(* IEC 61131-3 sources: RegAx/test, 7 files *)

(* ---- Assert.st ---- *)
USING AxUnit.ResultFunctions;
USING System.Strings;

NAMESPACE AxUnit.Assert

    /// Succeeds when the provided condition is TRUE.
    FUNCTION PUBLIC IsTrue
        VAR_INPUT
            /// Condition that must evaluate to TRUE.
            condition : BOOL;
        END_VAR
        IF condition THEN
            axunit_Succeed();
        ELSE
            axunit_Fail('Condition is not true');
        END_IF;
    END_FUNCTION

    /// Succeeds when the provided condition is FALSE.
    FUNCTION PUBLIC IsFalse
        VAR_INPUT
            /// Condition that must evaluate to FALSE.
            condition : BOOL;
        END_VAR
        IF NOT condition THEN
            axunit_Succeed();
        ELSE
            axunit_Fail('Condition is not false');
        END_IF;
    END_FUNCTION

END_NAMESPACE

(* ---- TestRegexClasses.st ---- *)
USING AxUnit.Assert;
USING Simatic.Ax.RegAx;
NAMESPACE RegexTests

    {TestFixture}
    /// Verifies shorthand character classes like \d and \w.
    CLASS TestRegexClasses
        VAR
            /// Regex instance reused across class test cases.
            _regex : Regex;
        END_VAR

        {Test}
        /// Ensures one or more digits are matched by \d+.
        METHOD PUBLIC Matches_Digit_Class_With_Plus
            _regex.SetPattern('^\d+$$');
            _regex.SetInput('12345');

            IsTrue(_regex.Match());
            Equal(expected := '12345', actual := _regex.GetMatch());
        END_METHOD

        {Test}
        /// Ensures \d+ rejects inputs containing letters.
        METHOD PUBLIC Rejects_Digit_Class_When_Letters_Appear
            _regex.SetPattern('^\d+$$');
            _regex.SetInput('123a');

            IsFalse(_regex.Match());
        END_METHOD

        {Test}
        /// Ensures \w works together with a bounded range quantifier.
        METHOD PUBLIC Matches_Word_Class_With_Range_Quantifier
            _regex.SetPattern('^\w{3,5}$$');
            _regex.SetInput('ab_9');

            IsTrue(_regex.Match());
            Equal(expected := 'ab_9', actual := _regex.GetMatch());
        END_METHOD

        {Test}
        /// Ensures \w range quantifiers reject inputs below the minimum length.
        METHOD PUBLIC Rejects_Word_Class_When_Too_Short
            _regex.SetPattern('^\w{3,5}$$');
            _regex.SetInput('ab');

            IsFalse(_regex.Match());
        END_METHOD

        {Test}
        /// Ensures mixed alphabetic ranges like [a-zA-Z] match upper and lower case letters.
        METHOD PUBLIC Matches_Alphabetic_Character_Class_Range
            _regex.SetPattern('^[a-zA-Z]+$$');
            _regex.SetInput('AbCdEf');

            IsTrue(_regex.Match());
            Equal(expected := 'AbCdEf', actual := _regex.GetMatch());
        END_METHOD
    END_CLASS

END_NAMESPACE

(* ---- TestRegexEscapes.st ---- *)
USING AxUnit.Assert;
USING Simatic.Ax.RegAx;
USING System.Strings;
NAMESPACE RegexTests

    {TestFixture}
    /// Verifies escaped literals and IP-like matching scenarios.
    CLASS TestRegexEscapes
        VAR
            /// Regex instance reused across escape and IP test cases.
            _regex : Regex;
        END_VAR

        /// Returns the substring after the first occurrence of a separator.
        METHOD PRIVATE TailAfterFirstSeparator : STRING
            VAR_INPUT
                input : STRING;
                separator : CHAR;
            END_VAR
            VAR
                currentIndex : INT;
                inputLength : INT;
                result : STRING;
                separatorFound : BOOL;
            END_VAR

            result := '';
            inputLength := LengthOf(input);
            separatorFound := FALSE;

            FOR currentIndex := 1 TO inputLength DO
                IF separatorFound THEN
                    result := CONCAT(result, input[currentIndex]);
                ELSIF input[currentIndex] = separator THEN
                    separatorFound := TRUE;
                END_IF;
            END_FOR;

            TailAfterFirstSeparator := result;
        END_METHOD

        {Test}
        /// Ensures an escaped dot is treated as a literal dot.
        METHOD PUBLIC Matches_Escaped_Dot
            _regex.SetPattern('^\.$$');
            _regex.SetInput('.');

            IsTrue(_regex.Match());
            Equal(expected := '.', actual := _regex.GetMatch());
        END_METHOD

        {Test}
        /// Ensures a simple dotted digit pattern matches a typical IP-like string.
        METHOD PUBLIC Matches_Simple_Ip_Like_Pattern
            _regex.SetPattern('^\d{1,3}\.\d{1,3}\.\d{1,3}\.\d{1,3}$$');
            _regex.SetInput('192.168.0.1');

            IsTrue(_regex.Match());
            Equal(expected := '192.168.0.1', actual := _regex.GetMatch());
        END_METHOD

        {Test}
        /// Ensures the same IP-like pattern accepts minimum-width blocks.
        METHOD PUBLIC Matches_Simple_Ip_Like_Pattern_With_Min_Values
            _regex.SetPattern('^\d{1,3}\.\d{1,3}\.\d{1,3}\.\d{1,3}$$');
            _regex.SetInput('0.0.0.0');

            IsTrue(_regex.Match());
            Equal(expected := '0.0.0.0', actual := _regex.GetMatch());
        END_METHOD

        {Test}
        /// Ensures the same IP-like pattern accepts maximum-width blocks.
        METHOD PUBLIC Matches_Simple_Ip_Like_Pattern_With_Max_Width_Blocks
            _regex.SetPattern('^\d{1,3}\.\d{1,3}\.\d{1,3}\.\d{1,3}$$');
            _regex.SetInput('255.255.255.255');

            IsTrue(_regex.Match());
            Equal(expected := '255.255.255.255', actual := _regex.GetMatch());
        END_METHOD

        {Test}
        /// Ensures the regex checks structure only and not numeric IPv4 ranges.
        METHOD PUBLIC Matches_Simple_Ip_Like_Pattern_Even_When_Block_Value_Exceeds_Ipv4_Range
            _regex.SetPattern('^\d{1,3}\.\d{1,3}\.\d{1,3}\.\d{1,3}$$');
            _regex.SetInput('999.999.999.999');

            IsTrue(_regex.Match());
            Equal(expected := '999.999.999.999', actual := _regex.GetMatch());
        END_METHOD

        {Test}
        /// Ensures an unanchored IP-like pattern extracts only the IP part from a URL.
        METHOD PUBLIC Finds_Ip_Address_Inside_Url_And_Returns_Only_The_Ip
            _regex.SetPattern('\d{1,3}\.\d{1,3}\.\d{1,3}\.\d{1,3}');
            _regex.SetInput('http://192.168.0.1');

            IsTrue(_regex.Match());
            Equal(expected := '192.168.0.1', actual := _regex.GetMatch());
        END_METHOD

        {Test}
        /// Ensures an unanchored IP-like pattern extracts only the IP part from an HTTPS URL with a port.
        METHOD PUBLIC Finds_Ip_Address_Inside_Https_Url_With_Port_And_Returns_Only_The_Ip
            _regex.SetPattern('\d{1,3}\.\d{1,3}\.\d{1,3}\.\d{1,3}');
            _regex.SetInput('https://192.168.0.1:5050');

            IsTrue(_regex.Match());
            Equal(expected := '192.168.0.1', actual := _regex.GetMatch());
        END_METHOD

        {Test}
        /// Demonstrates manual iteration over successive IP blocks by advancing the remaining input.
        METHOD PUBLIC Finds_All_Ip_Blocks_By_Repeating_Single_Block_Match_On_Remaining_Input
            VAR
                remainingInput : STRING;
            END_VAR

            _regex.SetPattern('\d{1,3}');

            remainingInput := 'https://192.168.0.1';
            _regex.SetInput(remainingInput);
            IsTrue(_regex.Match());
            Equal(expected := '192', actual := _regex.GetMatch());

            remainingInput := THIS.TailAfterFirstSeparator(input := remainingInput, separator := '.');
            _regex.SetInput(remainingInput);
            IsTrue(_regex.Match());
            Equal(expected := '168', actual := _regex.GetMatch());

            remainingInput := THIS.TailAfterFirstSeparator(input := remainingInput, separator := '.');
            _regex.SetInput(remainingInput);
            IsTrue(_regex.Match());
            Equal(expected := '0', actual := _regex.GetMatch());

            remainingInput := THIS.TailAfterFirstSeparator(input := remainingInput, separator := '.');
            _regex.SetInput(remainingInput);
            IsTrue(_regex.Match());
            Equal(expected := '1', actual := _regex.GetMatch());
        END_METHOD

        {Test}
        /// Ensures MatchNext can iterate over all IP blocks without modifying the input string.
        METHOD PUBLIC Finds_All_Ip_Blocks_With_MatchNext
            _regex.SetPattern('\d{1,3}');
            _regex.SetInput('https://192.168.0.1');

            IsTrue(_regex.Match());
            Equal(expected := '192', actual := _regex.GetMatch());

            IsTrue(_regex.MatchNext());
            Equal(expected := '168', actual := _regex.GetMatch());

            IsTrue(_regex.MatchNext());
            Equal(expected := '0', actual := _regex.GetMatch());

            IsTrue(_regex.MatchNext());
            Equal(expected := '1', actual := _regex.GetMatch());

            IsFalse(_regex.MatchNext());
        END_METHOD

        {Test}
        /// Ensures MatchNext reports the positions of successive matches.
        METHOD PUBLIC Reports_Start_And_End_Index_For_Successive_MatchNext_Calls
            _regex.SetPattern('\d{1,3}');
            _regex.SetInput('https://192.168.0.1');

            IsTrue(_regex.Match());
            Equal(expected := '192', actual := _regex.GetMatch());
            Equal(expected := 9, actual := _regex.GetMatchStartIndex());
            Equal(expected := 11, actual := _regex.GetMatchEndIndex());

            IsTrue(_regex.MatchNext());
            Equal(expected := '168', actual := _regex.GetMatch());
            Equal(expected := 13, actual := _regex.GetMatchStartIndex());
            Equal(expected := 15, actual := _regex.GetMatchEndIndex());
        END_METHOD

        {Test}
        /// Ensures the IP-like pattern rejects inputs with a missing final block.
        METHOD PUBLIC Rejects_Simple_Ip_Like_Pattern_When_Last_Block_Missing
            _regex.SetPattern('^\d{1,3}\.\d{1,3}\.\d{1,3}\.\d{1,3}$$');
            _regex.SetInput('192.168.0');

            IsFalse(_regex.Match());
        END_METHOD

        {Test}
        /// Ensures the IP-like pattern rejects blocks longer than three digits.
        METHOD PUBLIC Rejects_Simple_Ip_Like_Pattern_When_Block_Is_Too_Long
            _regex.SetPattern('^\d{1,3}\.\d{1,3}\.\d{1,3}\.\d{1,3}$$');
            _regex.SetInput('1234.168.0.1');

            IsFalse(_regex.Match());
        END_METHOD

        {Test}
        /// Ensures the IP-like pattern rejects non-digit characters inside a block.
        METHOD PUBLIC Rejects_Simple_Ip_Like_Pattern_When_Non_Digit_Appears_In_Block
            _regex.SetPattern('^\d{1,3}\.\d{1,3}\.\d{1,3}\.\d{1,3}$$');
            _regex.SetInput('192.16a.0.1');

            IsFalse(_regex.Match());
        END_METHOD

        {Test}
        /// Ensures the IP-like pattern rejects wrong separators.
        METHOD PUBLIC Rejects_Simple_Ip_Like_Pattern_When_Separator_Is_Wrong
            _regex.SetPattern('^\d{1,3}\.\d{1,3}\.\d{1,3}\.\d{1,3}$$');
            _regex.SetInput('192,168.0.1');

            IsFalse(_regex.Match());
        END_METHOD

        {Test}
        /// Ensures the IP-like pattern rejects trailing whitespace when anchored.
        METHOD PUBLIC Rejects_Simple_Ip_Like_Pattern_When_Whitespace_Is_Present
            _regex.SetPattern('^\d{1,3}\.\d{1,3}\.\d{1,3}\.\d{1,3}$$');
            _regex.SetInput('192.168.0.1 ');

            IsFalse(_regex.Match());
        END_METHOD

        {Test}
        /// Ensures the IP-like pattern rejects a leading separator.
        METHOD PUBLIC Rejects_Simple_Ip_Like_Pattern_When_Leading_Dot_Is_Present
            _regex.SetPattern('^\d{1,3}\.\d{1,3}\.\d{1,3}\.\d{1,3}$$');
            _regex.SetInput('.192.168.0.1');

            IsFalse(_regex.Match());
        END_METHOD

        {Test}
        /// Ensures the IP-like pattern rejects a trailing separator.
        METHOD PUBLIC Rejects_Simple_Ip_Like_Pattern_When_Trailing_Dot_Is_Present
            _regex.SetPattern('^\d{1,3}\.\d{1,3}\.\d{1,3}\.\d{1,3}$$');
            _regex.SetInput('192.168.0.1.');

            IsFalse(_regex.Match());
        END_METHOD
    END_CLASS

END_NAMESPACE

(* ---- TestRegexInvalidPatterns.st ---- *)
USING AxUnit.Assert;
USING Simatic.Ax.RegAx;

NAMESPACE RegexTests

    {TestFixture}
    /// Verifies that unsupported or malformed patterns are rejected safely.
    CLASS TestRegexInvalidPatterns
        VAR
            /// Regex instance reused across invalid-pattern test cases.
            _regex : Regex;
        END_VAR

        {Test}
        /// Ensures unsupported group syntax is rejected.
        METHOD PUBLIC Rejects_Unsupported_Group_Syntax
            _regex.SetPattern('^(ab)$$');
            _regex.SetInput('ab');

            IsFalse(_regex.Match());
        END_METHOD

        {Test}
        /// Ensures unsupported alternation syntax is rejected.
        METHOD PUBLIC Rejects_Unsupported_Alternation_Syntax
            _regex.SetPattern('^a|b$$');
            _regex.SetInput('a');

            IsFalse(_regex.Match());
        END_METHOD

        {Test}
        /// Ensures invalid quantifier ranges are rejected.
        METHOD PUBLIC Rejects_Invalid_Quantifier_Range
            _regex.SetPattern('^a{3,2}$$');
            _regex.SetInput('aaa');

            IsFalse(_regex.Match());
        END_METHOD

        {Test}
        /// Ensures dangling escape sequences are rejected.
        METHOD PUBLIC Rejects_Dangling_Escape
            _regex.SetPattern('abc\');
            _regex.SetInput('abc');

            IsFalse(_regex.Match());
        END_METHOD

        {Test}
        /// Ensures block-type patterns requiring groups and alternation remain unsupported.
        METHOD PUBLIC Rejects_Block_Type_Pattern_With_Group_And_Alternation
            _regex.SetPattern('(FB|OB|FC)[0-9]{1,5}');
            _regex.SetInput('ADD1@1_FC1.bin');

            IsFalse(_regex.Match());
        END_METHOD
    END_CLASS

END_NAMESPACE

(* ---- TestRegexLiterals.st ---- *)
USING AxUnit.Assert;
USING Simatic.Ax.RegAx;

NAMESPACE RegexTests

    {TestFixture}
    /// Verifies literal matching behavior for anchored and unanchored patterns.
    CLASS TestRegexLiterals
        VAR
            /// Regex instance reused across literal test cases.
            _regex : Regex;
        END_VAR

        {Test}
        /// Ensures an anchored literal matches the full input.
        METHOD PUBLIC Matches_Exact_Literal_With_Anchors
            _regex.SetPattern('^abc$$');
            _regex.SetInput('abc');

            IsTrue(_regex.Match());
            Equal(expected := 'abc', actual := _regex.GetMatch());
        END_METHOD

        {Test}
        /// Ensures an anchored literal is rejected when the input differs.
        METHOD PUBLIC Rejects_Exact_Literal_When_Input_Differs
            _regex.SetPattern('^abc$$');
            _regex.SetInput('abx');

            IsFalse(_regex.Match());
            Equal(expected := '', actual := _regex.GetMatch());
        END_METHOD

        {Test}
        /// Ensures an unanchored literal can be found inside a larger input.
        METHOD PUBLIC Finds_Unanchored_Literal_Inside_Input
            _regex.SetPattern('abc');
            _regex.SetInput('xxabczz');

            IsTrue(_regex.Match());
            Equal(expected := 'abc', actual := _regex.GetMatch());
        END_METHOD
    END_CLASS

END_NAMESPACE

(* ---- TestRegexQuantifiers.st ---- *)
USING AxUnit.Assert;
USING Simatic.Ax.RegAx;

NAMESPACE RegexTests

    {TestFixture}
    /// Verifies supported quantifiers like ?, *, and bounded repetitions.
    CLASS TestRegexQuantifiers
        VAR
            /// Regex instance reused across quantifier test cases.
            _regex : Regex;
        END_VAR

        {Test}
        /// Ensures an optional literal matches when the optional character is present.
        METHOD PUBLIC Matches_Optional_Literal_When_Present
            _regex.SetPattern('^colou?r$$');
            _regex.SetInput('colour');

            IsTrue(_regex.Match());
            Equal(expected := 'colour', actual := _regex.GetMatch());
        END_METHOD

        {Test}
        /// Ensures an optional literal matches when the optional character is absent.
        METHOD PUBLIC Matches_Optional_Literal_When_Absent
            _regex.SetPattern('^colou?r$$');
            _regex.SetInput('color');

            IsTrue(_regex.Match());
            Equal(expected := 'color', actual := _regex.GetMatch());
        END_METHOD

        {Test}
        /// Ensures exact repetition counts are accepted when the count matches.
        METHOD PUBLIC Matches_Exact_Repetition
            _regex.SetPattern('^a{3}$$');
            _regex.SetInput('aaa');

            IsTrue(_regex.Match());
            Equal(expected := 'aaa', actual := _regex.GetMatch());
        END_METHOD

        {Test}
        /// Ensures exact repetition counts reject shorter inputs.
        METHOD PUBLIC Rejects_Exact_Repetition_When_Count_Differs
            _regex.SetPattern('^a{3}$$');
            _regex.SetInput('aa');

            IsFalse(_regex.Match());
        END_METHOD

        {Test}
        /// Ensures open upper bound quantifiers accept longer runs.
        METHOD PUBLIC Matches_Open_Upper_Bound_Quantifier
            _regex.SetPattern('^a{2,}$$');
            _regex.SetInput('aaaa');

            IsTrue(_regex.Match());
            Equal(expected := 'aaaa', actual := _regex.GetMatch());
        END_METHOD

        {Test}
        /// Ensures the star quantifier accepts repeated middle literals.
        METHOD PUBLIC Matches_Star_Quantifier
            _regex.SetPattern('^ab*c$$');
            _regex.SetInput('abbbc');

            IsTrue(_regex.Match());
            Equal(expected := 'abbbc', actual := _regex.GetMatch());
        END_METHOD
    END_CLASS

END_NAMESPACE

(* ---- TestRegexRealWorldExamples.st ---- *)
USING AxUnit.Assert;
USING Simatic.Ax.RegAx;

NAMESPACE RegexTests

    {TestFixture}
    /// Verifies practical regex scenarios using the supported feature subset.
    CLASS TestRegexRealWorldExamples
        VAR
            /// Regex instance reused across real-world example test cases.
            _regex : Regex;
        END_VAR

        {Test}
        /// Ensures a simple department mailbox pattern with fixed local-part length matches.
        METHOD PUBLIC Matches_Corporate_Email_Address
            _regex.SetPattern('^[a-z]{4}@[a-z]{7}\.[a-z]{2}$$');
            _regex.SetInput('team@factory.de');

            IsTrue(_regex.Match());
            Equal(expected := 'team@factory.de', actual := _regex.GetMatch());
        END_METHOD

        {Test}
        /// Ensures the same email pattern rejects addresses without a top-level domain.
        METHOD PUBLIC Rejects_Email_Address_Without_Top_Level_Domain
            _regex.SetPattern('^[\w]+@[\w]+\.[a-z]{2,3}$$');
            _regex.SetInput('john_doe@factory');

            IsFalse(_regex.Match());
        END_METHOD

        {Test}
        /// Ensures a machine tag with a fixed prefix and four digits is accepted.
        METHOD PUBLIC Matches_Machine_Tag_With_Fixed_Prefix
            _regex.SetPattern('^MCH-\d{4}$$');
            _regex.SetInput('MCH-2048');

            IsTrue(_regex.Match());
            Equal(expected := 'MCH-2048', actual := _regex.GetMatch());
        END_METHOD

        {Test}
        /// Ensures a machine tag is rejected when the numeric part is too short.
        METHOD PUBLIC Rejects_Machine_Tag_When_Digit_Count_Is_Too_Short
            _regex.SetPattern('^MCH-\d{4}$$');
            _regex.SetInput('MCH-248');

            IsFalse(_regex.Match());
        END_METHOD

        {Test}
        /// Ensures a semantic version string with three numeric blocks matches.
        METHOD PUBLIC Matches_Semantic_Version_String
            _regex.SetPattern('^\d+\.\d+\.\d+$$');
            _regex.SetInput('2.14.7');

            IsTrue(_regex.Match());
            Equal(expected := '2.14.7', actual := _regex.GetMatch());
        END_METHOD

        {Test}
        /// Ensures a semantic version string is rejected when a block is missing.
        METHOD PUBLIC Rejects_Semantic_Version_When_Patch_Block_Is_Missing
            _regex.SetPattern('^\d+\.\d+\.\d+$$');
            _regex.SetInput('2.14');

            IsFalse(_regex.Match());
        END_METHOD

        {Test}
        /// Ensures a CSV-like sensor record with three numeric fields matches.
        METHOD PUBLIC Matches_Sensor_Record_With_Comma_Separated_Numbers
            _regex.SetPattern('^\d+,\d+,\d+$$');
            _regex.SetInput('120,45,998');

            IsTrue(_regex.Match());
            Equal(expected := '120,45,998', actual := _regex.GetMatch());
        END_METHOD

        {Test}
        /// Ensures a CSV-like sensor record rejects alphabetic noise in a field.
        METHOD PUBLIC Rejects_Sensor_Record_When_Field_Contains_Letters
            _regex.SetPattern('^\d+,\d+,\d+$$');
            _regex.SetInput('120,4A,998');

            IsFalse(_regex.Match());
        END_METHOD

        {Test}
        /// Ensures a lowercase file name with a three-letter extension matches.
        METHOD PUBLIC Matches_Lowercase_File_Name_With_Extension
            _regex.SetPattern('^[a-z]+\.[a-z]{3}$$');
            _regex.SetInput('report.csv');

            IsTrue(_regex.Match());
            Equal(expected := 'report.csv', actual := _regex.GetMatch());
        END_METHOD

        {Test}
        /// Ensures a file name is rejected when the extension length is wrong.
        METHOD PUBLIC Rejects_File_Name_When_Extension_Length_Is_Wrong
            _regex.SetPattern('^[a-z]+\.[a-z]{3}$$');
            _regex.SetInput('report.xlsx');

            IsFalse(_regex.Match());
        END_METHOD

        {Test}
        /// Ensures a log level prefix can be found inside a log line.
        METHOD PUBLIC Finds_Log_Level_Inside_Log_Line
            _regex.SetPattern('\[[A-Z]{4,5}\]');
            _regex.SetInput('2026-07-16 [ERROR] Motor overload detected');

            IsTrue(_regex.Match());
            Equal(expected := '[ERROR]', actual := _regex.GetMatch());
        END_METHOD

        {Test}
        /// Ensures a PLC variable name with underscores and digits matches.
        METHOD PUBLIC Matches_Plc_Variable_Name
            _regex.SetPattern('^[A-Za-z_][A-Za-z0-9_]{3,15}$$');
            _regex.SetInput('Motor_01_Run');

            IsTrue(_regex.Match());
            Equal(expected := 'Motor_01_Run', actual := _regex.GetMatch());
        END_METHOD

        {Test}
        /// Ensures a PLC variable name is rejected when it starts with a digit.
        METHOD PUBLIC Rejects_Plc_Variable_Name_Starting_With_Digit
            _regex.SetPattern('^[A-Za-z_][A-Za-z0-9_]{3,15}$$');
            _regex.SetInput('1Motor_Run');

            IsFalse(_regex.Match());
        END_METHOD

        {Test}
        /// Ensures an HTTP endpoint with a fixed-shape host and numeric port matches.
        METHOD PUBLIC Matches_Http_Url_With_Port
            _regex.SetPattern('^http://plc\d{2}\.local:\d{4}$$');
            _regex.SetInput('http://plc01.local:8080');

            IsTrue(_regex.Match());
            Equal(expected := 'http://plc01.local:8080', actual := _regex.GetMatch());
        END_METHOD

        {Test}
        /// Ensures an HTTP URL is rejected when the port is missing.
        METHOD PUBLIC Rejects_Http_Url_When_Port_Is_Missing
            _regex.SetPattern('^http://[\w]+\.local:\d{4}$$');
            _regex.SetInput('http://plc01.local');

            IsFalse(_regex.Match());
        END_METHOD
    END_CLASS

END_NAMESPACE
